{attribute 'GeneratedUsingTerminal: EK1100-0000-0018'}
{attribute addProperty BoxType "EK1100-0000-0018"}
{attribute addProperty Id "A_0018_BK1250_0000_0019A_0018_BK1250_0000_0019_DD1CA4A70"}
{attribute addProperty CRC "145239466"}
{attribute addProperty Size "0"}
TYPE Term_23_EK1100_08A82DAA EXTENDS EK1100_1FC0878B :
STRUCT
	{attribute addProperty Name "A_0018_BK1250_0000_0019"}
	{attribute addProperty PreviousPort "Term 23 (EK1100) : B"}
	A_0018_BK1250_0000_0019 : A_0018_BK1250_0000_0019_DD1CA4A7;
END_STRUCT
END_TYPE

(* stored: Version 1.2.0.0, ProductVersion 3.1.4024.9
   DUT Term_23_EK1100_08A82DAA: Id {186b9d95-0b0d-44af-a134-596d17d5c3e4} *)
